KUKA KRL data list: B20_snh_global.dat

&ACCESS RV
&COMMENT V_1_0_0
DEFDAT B20_snh_global PUBLIC
;********************************
;Date: 20.12.2013
;Programmer: AIUT
;Description: Stud welding global positions
;********************************



ENDDAT
